{attribute 'qualified_only'}
VAR_GLOBAL
	FwLimit				AT	%I*	: ARRAY[1..GVL.axisNumMax] OF BOOL;		(*~ (OPC: 1 : available for OPC-clients) (OPC_PROP[0005]: 1 : OPC_PROP_RIGHTS, here read/write) *)
	BwLimit				AT  %I*	: ARRAY[1..GVL.axisNumMax] OF BOOL;		(*~ (OPC: 1 : available for OPC-clients) (OPC_PROP[0005]: 1 : OPC_PROP_RIGHTS, here read/write) *)
	
	coupledFwLimit		: ARRAY [1..GVL.axisNumMax] OF ARRAY [1..5] OF ST_MasterCoupling;	//Store for slave/master linking
	coupledBwLimit		: ARRAY [1..GVL.axisNumMax] OF ARRAY [1..5] OF ST_MasterCoupling;	//Store for slave/master linking

END_VAR

(* stored: Version 1.1.0.1, ProductVersion 3.1.4022.12
   GVL Limits: Id {bc15940f-38e2-463e-88a6-afd29e0a1edc} *)
